FUNCTION_BLOCK AdderTest IMPLEMENTS Testbench.IUnitTest
VAR
  _adder : Adder;
END_VAR

METHOD Test_Add_ReturnsCorrectResult
VAR_INPUT
  assertions : Testbench.IAssertions;
END_VAR
VAR
  result : INT;
END_VAR
// arrange

// act
result := _adder.AddInt(5, 3);

// assert
assertions.EqualsInt(8, result, 'Result is correct');
END_METHOD

END_FUNCTION_BLOCK

(* stored: Version 1.1.0.1, ProductVersion 3.1.4024.12
   POU AdderTest: Id {2cdb9ddd-ae20-45b5-b92a-76fc03bc0110}, SpecialFunc None
   Method Test_Add_ReturnsCorrectResult: Id {3e6190a4-8d03-4eb2-a842-0efcfc6fc15d} *)
